Fanuc KAREL source: kt00070.KL

-- PROVISIONAL review KL for V940-1; original PC SHA256 f6edb315049ab42435274e65667c074eccb6a53d347c685fa75dc56bc31c7cac
-- Incomplete behavior may be omitted. Consult companion uncertainty JSON. Do not deploy.
PROGRAM KT00070
%NOLOCKGROUP
VAR
  I1 : INTEGER
  OUT : REAL
-- UNRESOLVED_DECL Y2 type=002018
BEGIN
  -- V9_ZERO_TABLE_METADATA_HINT layout=0001; no indexed target words; source/name/runtime held
  -- UNRESOLVED_PC offsets 5-16; opcodes 2E,23
  -- UNRESOLVED_PC offsets 21-35; opcodes 2E,22,9D,33,B2
  -- UNRESOLVED_PC offsets 40-63; opcodes 21,22,9D,33,B1,54,64,23
  -- UNRESOLVED_PC offsets 68-72; opcodes 7F
END KT00070
